Universal Robots PolyScope program: Test Weld Peg Motion.urp

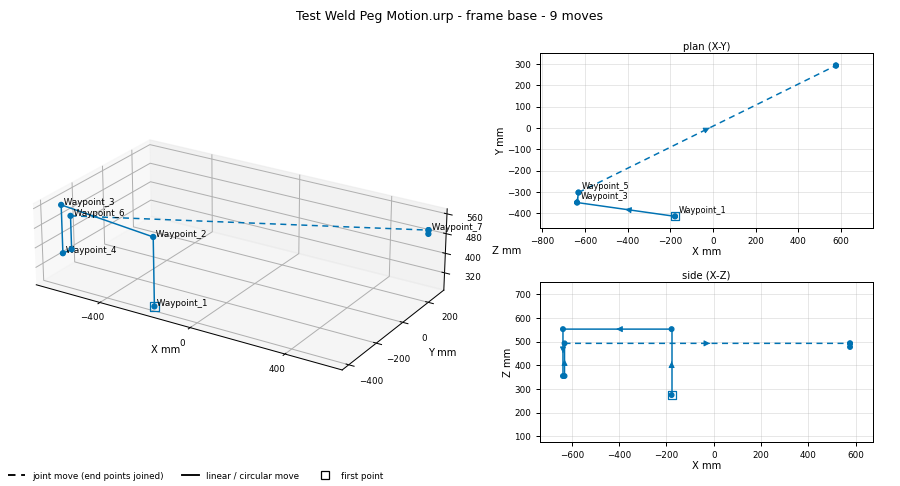
[picture p0: tool path of Test Weld Peg Motion.urp in frame base, 9 of 9 moves have a stored position in this frame; points joined in program order, loops and branches not executed]
Program Test Weld Peg Motion (installation=default directory=/programs createdIn=5.14.5 lastSavedIn=5.14.5 robotSerialNumber=20236801216)
Calibrated DH parameters: a=[-0.000021, -0.748897, -0.28186, -0.00004, -0.000055, 0]; d=[0.236225, -424.082933, -1564.66872, 1988.95162, 0.159094, 0.153873]; alpha=[1.570844, 0.001002, 0.000337, 1.571488, -1.569996, 0]; deltaTheta=[0, -0.516316, 5.626292, 1.173211, 0.000001, 0]
InitVariablesNode
Robot Program (runOnlyOnce=true)
  'Start Point: Home'
  MoveJ speed 60 deg/s, acceleration 80 deg/s^2 (useActiveTCP=true) feature=Base
    Waypoint Waypoint_1: TCP in base x=-178.197 y=-413.642 z=275.211 mm, rx=-0.1147 ry=3.0868 rz=-0.038 rad; joints [-88.065, -87.595, -159.71, -21.34, 93.022, -2.286] deg; TCP offset x=-0.005 y=-0.004 z=-0.034 mm, rx=0 ry=0 rz=0 rad
  MoveL speed 250 mm/s, acceleration 1200 mm/s^2 (useActiveTCP=true) feature=Base
    'Lift gun out of holder'
    Waypoint Waypoint_2: TCP in base x=-178.197 y=-413.594 z=553.617 mm, rx=-0.1147 ry=3.0867 rz=-0.0379 rad; joints [-88.047, -60.266, -142.398, -65.984, 93.01, -2.269] deg
    'Move to bucket'
    Waypoint Waypoint_3: TCP in base x=-637.123 y=-348.923 z=553.625 mm, rx=-0.1148 ry=3.0867 rz=-0.0379 rad; joints [-135.958, -85.087, -126.685, -59.573, 93.074, -50.247] deg
    Waypoint Waypoint_4: TCP in base x=-637.124 y=-348.923 z=355.419 mm, rx=-0.1147 ry=3.0867 rz=-0.038 rad; joints [-135.961, -96.884, -135.74, -38.721, 93.077, -50.246] deg
  'extrude out a foot'
  Wait Sleep waitTime=6
  MoveL speed 40 mm/s, acceleration 1200 mm/s^2 (useActiveTCP=true) feature=Base
    'slice over knife'
    Waypoint Waypoint_5: TCP in base x=-630.521 y=-301.963 z=355.442 mm, rx=-0.1147 ry=3.0868 rz=-0.038 rad; joints [-138.451, -95.206, -137.712, -38.557, 93.016, -52.74] deg
  MoveL speed 250 mm/s, acceleration 1200 mm/s^2 (useActiveTCP=true) feature=Base
    Waypoint Waypoint_6: TCP in base x=-630.515 y=-301.956 z=493.474 mm, rx=-0.1147 ry=3.0868 rz=-0.038 rad; joints [-138.448, -86.027, -131.576, -53.873, 93.012, -52.739] deg
  MoveJ speed 60 deg/s, acceleration 80 deg/s^2 (useActiveTCP=true) feature=Base
    'go to weld peg'
    Waypoint Waypoint_7: TCP in base x=575.58 y=292.976 z=493.476 mm, rx=-0.1148 ry=3.0867 rz=-0.0379 rad; joints [45.82, -81.467, -136.118, -51.256, 86.919, 131.536] deg
  MoveL speed 250 mm/s, acceleration 1200 mm/s^2 (useActiveTCP=true) feature=Base
    'tilt head'
    Waypoint Waypoint_8: TCP in base x=575.531 y=292.898 z=493.385 mm, rx=-0.0813 ry=2.3673 rz=-0.1895 rad; joints [54.38, -83.795, -145.713, -16.792, 50.925, 131.952] deg
    Waypoint Waypoint_9: TCP in base x=575.533 y=292.902 z=478.246 mm, rx=-0.0813 ry=2.3673 rz=-0.1895 rad; joints [54.379, -85.19, -146.444, -14.666, 50.926, 131.952] deg
  ''
  Wait Sleep waitTime=8
